(* PLC project Unnamed, Unknown Unnamed 1 *)
(* stored: creationDateTime 2026-02-02T16:50:47, modificationDateTime 2026-02-02T16:50:47 *)

CONFIGURATION Config0
  RESOURCE Res0 ON PLC
  END_RESOURCE
END_CONFIGURATION
